TYPE Vec7b : ARRAY[1..7] OF BOOl; END_TYPE

(* stored: Version 1.1.0.1, ProductVersion 3.1.4024.12
   DUT Vec7b: Id {8b0c0712-bfac-403c-a8c1-0d9d5f12c181} *)
